PROGRAM MAIN
VAR
END_VAR

PrgMqttCom();

END_PROGRAM

(* stored: Version 1.1.0.1, ProductVersion 3.1.4024.11
   POU MAIN: Id {c9aae06e-c2e5-4a02-96c5-f1337a91e27e}, SpecialFunc None *)
